VAR_OUTPUT
LampStop   :BOOL := FALSE; (* Флаг "Активен режим СТОП". *)
LampManual :BOOL := FALSE; (* Флаг "Активен РУЧНОЙ режим". *)
LampAuto   :BOOL := FALSE; (* Флаг "Активен АВТОМАТИЧЕСКИЙ режим. *)
END_VAR

VAR
State1    :INT  := 0    ; (* Локальный граф состояний. *)
FlagError :BOOL := FALSE; (* Флаг запрещенного состояния входов. *)
END_VAR

VAR CONSTANT
STATE_STOP   :INT := 0; (* Состояние "СТОП РЕЖИМ". *)
STATE_MANUAL :INT := 1; (* Состояние "РУЧНОЙ РЕЖИМ". *)
STATE_AUTO   :INT := 2; (* Состояние "АВТОМАТИЧЕСКИЙ РЕЖИМ". *)
END_VAR
(*
 Переключатель режимов работы.
          DbModeSelector
    +------------------------+
    |     FbModeSelector     |
 ->-|ButtonStop      LampStop|->-
 ->-|ButtonManual  LampManual|->-
 ->-|ButtonAuto      LampAuto|->-
   -|Error                   |
   -|Reset                   |
    +------------------------+
*)

(* Запрещенное состояние: *)
(* Если вместе с кнопкой стоп одновременно нажали еще что-то. *)
FlagError:=
((ButtonStop AND ButtonAuto) OR
( ButtonStop AND ButtonManual));

(* При перезагрузке контроллера режим СТОП. *)
IF (Reset OR FlagError) THEN
    State1     := STATE_STOP;
    LampStop   := TRUE;
    LampManual := FALSE;
    LampAuto   := FALSE;
ELSE
    (* Граф состояний. *)
    CASE State1 OF

    STATE_STOP: (* Режим СТОП. *)
    LampStop   := TRUE;
    LampManual := FALSE;
    LampAuto   := FALSE;
    (* Переход СТОП -> РУЧНОЙ. *)
    IF ButtonManual THEN
    State1     := STATE_MANUAL;
    LampStop   := FALSE;
    LampManual := TRUE;
    LampAuto   := FALSE;
    END_IF;
    (* Переход СТОП -> АВТОМАТ. *)
    IF (ButtonAuto AND NOT(Error)) THEN
    State1     := STATE_AUTO;
    LampStop   := FALSE;
    LampManual := FALSE;
    LampAuto   := TRUE;
    END_IF;

    STATE_MANUAL: (* Режим РУЧНОЙ. *)
    LampStop   := FALSE;
    LampManual := TRUE;
    LampAuto   := FALSE;
    (* Переход РУЧНОЙ -> СТОП. *)
    IF ButtonStop THEN
    State1     := 0;
    LampStop   := TRUE;
    LampManual := FALSE;
    LampAuto   := FALSE;
    END_IF;
    (* Преход РУЧНОЙ -> АВТОМАТ. *)
    IF (ButtonAuto AND NOT(Error)) THEN
    State1     := STATE_AUTO;
    LampStop   := FALSE;
    LampManual := FALSE;
    LampAuto   := TRUE;
    END_IF;

    STATE_AUTO: (* Режим АВТОМАТ. *)
    LampStop   := FALSE;
    LampManual := FALSE;
    LampAuto   := TRUE;
    (* Переход АВТОМАТ -> СТОП. *)
    IF (ButtonStop OR Error) THEN
    State1     := STATE_STOP;
    LampStop   := TRUE;
    LampManual := FALSE;
    LampAuto   := FALSE;
    END_IF;
    (* Переход АВТОМАТ -> РУЧНОЙ. *)
    IF ButtonManual THEN
    State1     := STATE_MANUAL;
    LampStop   := FALSE;
    LampManual := TRUE;
    LampAuto   := FALSE;
    END_IF;

    ELSE (*СТОП при неопределенном состоянии. *)
    State1 := STATE_STOP;
    END_CASE;

END_IF; (* IF (Reset OR FlagError) THEN *)

(*
 Граф состояний.

 Если ошибка Error активна можно работать только в ручном режиме.
 Reset должен срабатывать при перезагрузке или включении питания.

                                  |
                                 -+-Reset OR FlagError
                                  |
                                  V
                        +-------------------+
                        | State1 =          |
            +---------->| STATE_STOP        |-----------+
            |           | LampStop = 1      |           |
            |           +-------------------+           |
            |                |         ^                |
            |                |         |                |
            |   ButtonManual-+-       -+-ButtonStop     |
            |                |         |                |
            |                V         |                |
            |           +-------------------+           |
 ButtonStop |           | State1 =          |           | ButtonAuto
        OR -+-          | STATE_MANUAL      |          -+- AND
      Error |           | LampManual = 1    |           | NOT(Error)
            |           +-------------------+           |
            |                |         ^                |
            |     ButtonAuto |         |                |
            |           AND -+-       -+-ButtonManual   |
            |     NOT(Error) |         |                |
            |                V         |                |
            |           +-------------------+           |
            |           | State1 =          |           |
            +-----------| STATE_AUTO        |<----------+
                        | LampAuto = 1      |
                        +-------------------+

 Пример организации интерфейса пользователя для HMI.
 При нажатии кнопоки AUTO тег ButtonAuto = 1.
 В автоматическом режиме работы тег LampAuto = 1 дает эффект нажатия на кнопку AUTO.
 Кнопки MANUAL, STOP работают аналогично.
 Так как кнопки без фиксации то можно параллельно кнопкам на экране подключать физические кнопки.

 +--------------------------------------------------------+
 | MENU: "Errors"                                         |
 +--------------------------------------------------------+
 | 0. No Error (OK).                                      |
 |                                                        |
 |                                                        |
 |                                                        |
 |                                                        |
 |                                                        |
 |                                                        |
 +--------------------------------------------------------+
 | +--------+ +--------+ +--------+ +--------+ +--------+ |
 | | < MENU | |  AUTO  | | MANUAL | |  STOP  | | MENU > | |
 | +--------+ +--------+ +--------+ +--------+ +--------+ |
 +--------------------------------------------------------+

@COPYLEFT ALL WRONGS RESERVED :)
Author: VA
Contacts: DIY.PLC.314@gmail.com
Date start LIB_PLC: 2014
License: GNU GPL-2.0-or-later
https://www.gnu.org/licenses/old-licenses/gpl-2.0.html
https://www.youtube.com/watch?v=n1F_MfLRlX0
https://www.youtube.com/@DIY_PLC
https://github.com/DIYPLC/LIB_PLC
https://oshwlab.com/diy.plc.314/PLC_HW1_SW1
https://3dtoday.ru/3d-models/mechanical-parts/body/korpus-na-din-reiku
https://t.me/DIY_PLC
*)
END_FUNCTION_BLOCK

(* POU LIB_PLC/FbMotor, ST *)
FUNCTION_BLOCK FbMotor (* Двигатель с частотником и контактором. *)

VAR_INPUT
MotorRun       :BOOL := FALSE; (* Команда: включить двигатель. *)
VoltageOk      :BOOL := FALSE; (* Схема собрана 380VAC Ok. *)
DriveOk        :BOOL := FALSE; (* Обратная связь: нет ошибок на частотном приводе. *)
ContactorOk    :BOOL := FALSE; (* Обратная связь: контактор включился. *)
TimeMonitoring :DINT := 1000 ; (* Время гарантированного включения контактора [мс]. *)
TimeDelayOn    :DINT := 1000 ; (* Время задержки включения частотника [мс]. *)
TimeDelayOff   :DINT := 5000 ; (* Время задержки выключения контактора [мс]. *)
Ts_ms          :DINT := 100  ; (* Шаг дискретизации по времени [мс]. *)
Reset          :BOOL := FALSE; (* Сброс при перезагрузке. *)
END_VAR

VAR_OUTPUT
MotorOn        :BOOL := FALSE; (* Включить двигатель. *)
ContactorOn    :BOOL := FALSE; (* Включить контактор. *)
ErrorVoltage   :BOOL := FALSE; (* Схема разобрана нет 380VAC. *)
ErrorDrive     :BOOL := FALSE; (* Ошибка частотного привода. *)
ErrorContactor :BOOL := FALSE; (* Ошибка контактора. *)
END_VAR

VAR
State1 :INT  := 0; (* Граф сосояния частотника и контактора. *)
Timer1 :DINT := 0; (* Таймер для задержки переключения между частотником и контактором [мс]. *)
Timer2 :DINT := 0; (* Таймер для формирования ошибки контактора [мс]. *)
END_VAR

VAR CONSTANT
STATE_STOP          :INT := 0; (* Состояние "Стоп". *)
STATE_CONTACTOR_ON  :INT := 1; (* Состояние "Включение контактора". *)
STATE_DRIVE_ON      :INT := 2; (* Состояние "Включение частотного привода". *)
STATE_RUN           :INT := 3; (* Состояние "Работа". *)
STATE_DRIVE_OFF     :INT := 4; (* Состояние "Выключение частотного привода". *)
STATE_CONTACTOR_OFF :INT := 5; (* Состояние "Выключение контактора". *)
END_VAR
(*
 Двигатель с частотником и контактором.
                 DbMotor
    +-------------------------------+
    |            FbMotor            |
 ->-|MotorRun                MotorOn|->-
   -|VoltageOk           ContactorOn|-
   -|DriveOk            ErrorVoltage|-
   -|ContactorOk          ErrorDrive|-
   -|TimeMonitoring   ErrorContactor|-
   -|TimeDelayOn                    |
   -|TimeDelayOff                   |
   -|Ts_ms                          |
   -|Reset                          |
    +-------------------------------+
*)

(* Схема разобрана нет 380VAC. *)
ErrorVoltage := NOT(VoltageOk);

(* Ошибка частотного привода. *)
ErrorDrive := NOT(DriveOk);

(* Формируем ошибку контактора. *)
(* Контактор включается не сразу. *)
(* За время TimeMonitoring контактор обязан включиться, иначе ошибка. *)
(* Так же следим чтобы контактор выключился и контакты не залипли. *)
IF (ContactorOn) THEN
(* Следим чтобы контактор вовремя включился. *)
  IF (ContactorOk) THEN
  (* Контактор включился. *)
  Timer2 := 0;
  ErrorContactor := FALSE;
  ELSE
    IF (Timer2 <= TimeMonitoring) THEN
    (* Контактор еще не включился. *)
    Timer2 := Timer2 + Ts_ms;
    ErrorContactor := FALSE;
    ELSE
    (* Ошибка контактор не включился за время TimeMonitoring *)
    ErrorContactor := TRUE;
    END_IF;
  END_IF;
ELSE
(* Следим чтобы контактор вовремя выключился. *)
  IF NOT(ContactorOk) THEN
  (* Контактор выключился. *)
  Timer2 := 0;
  ErrorContactor := FALSE;
  ELSE
    IF (Timer2 <= TimeMonitoring) THEN
    (* Контактор еще не выключился. *)
    Timer2 := Timer2 + Ts_ms;
    ErrorContactor := FALSE;
    ELSE
    (* Ошибка контактор не выключился за время TimeMonitoring *)
    ErrorContactor := TRUE;
    END_IF;
  END_IF;
END_IF;

(* Сброс при перезагрузке или ошибке. *)
IF (Reset OR ErrorVoltage OR ErrorDrive) THEN
State1 := STATE_STOP;
END_IF;

(* При включении двигателя должен сначала включиться контактор затем частотный привод. *)
(* При выключении двигателя должен сначала выключиться частотный привод, а затем контактор. *)
(* Это необходимо для увеличения времени жизни контактора. *)
(* Граф состояний. *)
CASE State1 OF

(* Состояние "Стоп". *)
STATE_STOP:
MotorOn     := FALSE;
ContactorOn := FALSE;
Timer1 := 0;
(* Если получили разрешение на включение то включаем контактор. *)
IF (MotorRun) THEN
State1 := STATE_CONTACTOR_ON;
END_IF;

(* Состояние "Включение контактора". *)
STATE_CONTACTOR_ON:
MotorOn     := FALSE;
ContactorOn := TRUE;
Timer1 := Timer1 + Ts_ms;
(* Перед включением частотника делаем паузу чтоб контактор успел включиться. *)
IF (Timer1 >= TimeDelayOn) THEN
State1 := STATE_DRIVE_ON;
END_IF;

(* Состояние "Включение частотного привода". *)
STATE_DRIVE_ON:
MotorOn     := TRUE;
ContactorOn := TRUE;
Timer1 := 0;
State1 := STATE_RUN;

(* Состояние "Работа". *)
STATE_RUN:
MotorOn     := TRUE;
ContactorOn := TRUE;
Timer1 := 0;
(* Если пришла команда выключить двигатель то сначала выключаем частотник. *)
IF NOT(MotorRun) THEN
State1 := STATE_DRIVE_OFF;
END_IF;

(* Состояние "Выключение частотного привода". *)
STATE_DRIVE_OFF:
MotorOn     := FALSE;
ContactorOn := TRUE;
Timer1 := Timer1 + Ts_ms;
(* Перед выключением контактора делаем паузу чтоб выключится без нагрузки. *)
IF (Timer1 >= TimeDelayOff) THEN
State1 := STATE_CONTACTOR_OFF;
END_IF;

(* Состояние "Выключение контактора". *)
STATE_CONTACTOR_OFF:
MotorOn     := FALSE;
ContactorOn := FALSE;
Timer1 := 0;
(* Переходим в состояние стоп. *)
State1 := STATE_STOP;

(* СТОП при неопределенном состоянии. *)
ELSE
State1 := STATE_STOP;
END_CASE;

(*
 Схема подключения блока FbMotor.

                +-------------------+
                | 380 VAC           |
                +-------------------+
                          |
                          v
                +-------------------+
                | Вводной автомат   |--> VoltageOk
                +-------------------+
                          |
                          v
                +-------------------+
     MotorOn -->| Частотный привод  |--> DriveOk
                +-------------------+
                          |
                          v
                +-------------------+
 ContactorOn -->| Контактор         |--> ContactorOk
                +-------------------+
                          |
                          v
                +-------------------+
                | Двигатель         |
                +-------------------+

@COPYLEFT ALL WRONGS RESERVED :)
Author: VA
Contacts: DIY.PLC.314@gmail.com
Date start LIB_PLC: 2014
License: GNU GPL-2.0-or-later
https://www.gnu.org/licenses/old-licenses/gpl-2.0.html
https://www.youtube.com/watch?v=n1F_MfLRlX0
https://www.youtube.com/@DIY_PLC
https://github.com/DIYPLC/LIB_PLC
https://oshwlab.com/diy.plc.314/PLC_HW1_SW1
https://3dtoday.ru/3d-models/mechanical-parts/body/korpus-na-din-reiku
https://t.me/DIY_PLC
*)
END_FUNCTION_BLOCK

(* POU LIB_PLC/FbPIDstep, ST *)
FUNCTION_BLOCK FbPIDstep (* ПИД-регулятор с двумя дискретными выходами. *)

VAR_INPUT
	PV       :REAL := 0.0  ; (* Измеренное значение регулируемого параметра 0...100[%]. *)
	SP       :REAL := 0.0  ; (* Заданное значение регулируемого параметра 0...100[%]. *)
	COM_RST  :BOOL := FALSE; (* Полная перезагрузка. *)
	LMNR_HS  :BOOL := FALSE; (* Датчик обранной связи клапан открыт. *)
	LMNR_LS  :BOOL := FALSE; (* Датчик обранной связи клапан закрыт. *)
	LMNS_ON  :BOOL := FALSE; (* Включить ружной режим управления. *)
	LMNUP    :BOOL := FALSE; (* Команда открыть в ручном режиме. *)
	LMNDN    :BOOL := FALSE; (* Команда закрыть в ручном режиме. *)
	GAIN     :REAL := 2.0  ; (* Пропорциональное усиление ошибки регулирования. *)
	TI       :REAL := 20.0 ; (* Время интегрирования [с]. *)
	DEADB_W  :REAL := 0.5  ; (* Зона нечувствительности к ошибке регулирования [%]. *)
	PULSE_TM :REAL := 1.0  ; (* Минимальное время выходного импульса [с]. *)
	BREAK_TM :REAL := 1.0  ; (* Минимально время между выходными импульсами [с]. *)
	MTR_TM   :REAL := 55.0 ; (* Время открытия исполнительного механизма с 0 до 100 [с]. *)
	DISV     :REAL := 0.0  ; (* Возмущающее воздействие к ошибке регулирования [%]. *)
	CYCLE    :REAL := 0.1  ; (* Шаг дискретизации по времени [с]. *)
END_VAR

VAR_OUTPUT
	QLMNUP :BOOL :=  FALSE; (* Открыть задвижку. *)
	QLMNDN :BOOL :=  FALSE; (* Закрыть задвижку. *)
END_VAR

VAR
	ER          :REAL := 0.0  ; (* Ошибка регулирования [%]. *)
	LMNRS_ON    :BOOL := FALSE; (* *)
	LMNRSVAL    :REAL := 0.0  ; (* *)
	LMNR_SIM    :REAL := 0.0  ; (* *)
	sFbPVal     :REAL := 0.0  ; (* Меняется во время регулирования. *)
	sThrOn      :REAL := 0.0  ; (* Иногда меняется во время регулирования (похоже на адаптивный гистерезис). *)
	siImpAus    :INT  := 0    ; (* -100...0...+100 *)
	stImpDauer  :REAL := 0.0  ; (* *)
	stPausDauer :REAL := 0.0  ; (* *)
END_VAR

VAR_TEMP
	Hvar     :REAL := 0.0 ; (* Вспомогательная переменная *)
	ErKp     :REAL := 0.0 ; (* Вспомогательная переменная *)
	rTi      :REAL := 0.0 ; (* Время интегрирования в real !!! не удалять !!! *)
	AdapIn1  :REAL := 0.0 ; (* Eingang 1 der Adaption der Ansprechschwelle *)
	AdapIn2  :REAL := 0.0 ; (* Eingang 2 der Adaption der Ansprechschwelle *)
	iImpEin  :INT  := 0   ; (* Eingang des Impulsformers *)
	rThrOff  :REAL := 0.0 ; (* Abschaltschwelle *)
	dInteg   :REAL := 0.0 ; (* Eingang des Integrierers in der Rückführung *)
	dThrStIn :REAL := 0.0 ; (* Three - step element input *)
	LmnrSim  :REAL := 0.0 ; (* Simulierte Stellungsrückmeldung *)
END_VAR
(*
 ПИД-регулятор с двумя дискретными выходами.
             DbPIDstep
    +-------------------------+
    |        FbPIDstep        |
 ->-|PV                 QLMNUP|->-
   -|SP                 QLMNDN|->-
   -|COM_RST                  |
   -|LMNR_HS                  |
   -|LMNR_LS                  |
   -|LMNS_ON                  |
   -|LMNUP                    |
   -|LMNDN                    |
   -|GAIN                     |
   -|TI                       |
   -|DEADB_W                  |
   -|PULSE_TM                 |
   -|BREAK_TM                 |
   -|MTR_TM                   |
   -|DISV                     |
   -|CYCLE                    |
    +-------------------------+
*)

IF COM_RST
THEN 
    LMNR_SIM    := LMNRSVAL;
    QLMNUP      := 0       ;
    QLMNDN      := 0       ;
    PV          := 0.0     ;
    ER          := 0.0     ;
    LMNRS_ON    := 0       ;
    LMNRSVAL    := 0.0     ;
    LMNR_SIM    := 0.0     ;
    sFbPVal     := 0.0     ;
    sThrOn      := 0.0     ;
    siImpAus    := 0       ;
    stImpDauer  := 0.0     ;
    stPausDauer := 0.0     ;
ELSE
    ErKp := SP - PV;
    IF    ErKp < ( -DEADB_W) THEN  ER := ErKp + DEADB_W;
    ELSIF ErKp > DEADB_W      THEN  ER := ErKp - DEADB_W;
    ELSE  ER := 0.0; END_IF;
    ErKp := ER * GAIN;
    rTi := TI;
    IF rTi < CYCLE * 0.5 THEN rTi := CYCLE * 0.5; END_IF; 
    Hvar := rTi - ABS(0.01 * ErKp * MTR_TM);
    IF Hvar < (rTi * 0.1)THEN rTi := rTi * 0.1; ELSE rTi := Hvar; END_IF;
    IF LMNS_ON 
    THEN 
        sFbPVal := 0.0;
    ELSE  
        IF siImpAus <> 0 
        THEN  
            dInteg := DINT_TO_REAL(INT_TO_DINT(siImpAus)) * CYCLE / MTR_TM;
        ELSE 
            IF (ErKp > 0.0 AND LMNR_HS) OR (ErKp < 0.0 AND LMNR_LS) OR (TI = 0.0)
            THEN 
                dInteg := 0.0;
            ELSE    
                dInteg  := (-ErKp) * CYCLE / rTi;
            END_IF;
        END_IF;
        sFbPVal := sFbPVal + dInteg;
        IF TI = 0.0
        THEN  
            IF    sFbPVal > 100.0 THEN sFbPVal := 100.0;
            ELSIF sFbPVal < 0.0   THEN sFbPVal := 0.0;
            END_IF;
        END_IF;
    END_IF;
    dThrStIn := ErKp - sFbPVal + DISV;
    AdapIn1 := ErKp;
    AdapIn2 := sFbPVal;
    rThrOff := 55.0 / MTR_TM * CYCLE;
    IF PULSE_TM > CYCLE
    THEN
    Hvar := PULSE_TM;
    ELSE
    Hvar := CYCLE;
    END_IF;
    Hvar := 100.0 * Hvar / MTR_TM;
    IF NOT(LMNR_HS OR LMNR_LS)
    THEN
        IF NOT (QLMNUP OR QLMNDN)
        THEN
            IF TI <> 0.0
            THEN
                IF ABS(AdapIn1) < ABS(AdapIn2)
                THEN
                    sThrOn := AdapIn1;
                ELSE
                    sThrOn := AdapIn2; 
                END_IF;
            ELSE
                IF PV = 0.0
                THEN
                    sThrOn := Hvar;
                ELSE 
                    sThrOn := ABS(ErKp) * 0.5;
                END_IF;
            END_IF;
            IF sThrOn > 10.0 THEN sThrOn := 10.0; END_IF;
            IF sThrOn < Hvar THEN sThrOn := Hvar; END_IF;
        END_IF;
    ELSE
        sThrOn := Hvar;
    END_IF;
    IF (siImpAus = 100 AND dThrStIn > rThrOff) OR (dThrStIn >= sThrOn)             THEN iImpEin := 100;
    ELSIF (siImpAus = -100 AND dThrStIn < ( -rThrOff)) OR (dThrStIn <= ( -sThrOn)) THEN iImpEin := -100;
    ELSE                                                                                iImpEin := 0;
    END_IF;
    IF LMNS_ON
    THEN
        IF LMNUP XOR LMNDN
        THEN
            IF LMNUP
            THEN
                iImpEin := 100;
            ELSE
                iImpEin := -100;
            END_IF;
        ELSE
            iImpEin := 0;
        END_IF;
    END_IF;
    IF (iImpEin = 100 AND LMNR_HS) OR (iImpEin = -100 AND LMNR_LS) THEN iImpEin := 0; END_IF;
    IF (siImpAus = -100 AND iImpEin = 100) OR (siImpAus = 100 AND iImpEin = -100)THEN iImpEin := 0; END_IF;
    IF siImpAus <> iImpEin
    THEN
        IF iImpEin = 0
        THEN
            IF stImpDauer <= 0.0
            THEN 
                siImpAus := 0;
                stPausDauer := BREAK_TM;
            END_IF;
        ELSE
            siImpAus := iImpEin;
            stImpDauer := PULSE_TM;
        END_IF;
    END_IF;
    IF stImpDauer > 0.0
    THEN
    stImpDauer := stImpDauer - CYCLE;
    ELSE
    stImpDauer := 0.0;
    END_IF;
    IF stPausDauer > 0.0
    THEN
    stPausDauer := stPausDauer - CYCLE;
    ELSE
    stPausDauer := 0.0;
    END_IF;
    IF ((siImpAus = 100) AND LMNR_HS) OR ((siImpAus = -100) AND LMNR_LS)
    THEN 
      siImpAus := 0;
      stImpDauer := 0.0;
    END_IF;
    IF NOT LMNRS_ON
    THEN
        LmnrSim := LMNRSVAL;
    ELSE
        LmnrSim := DINT_TO_REAL(INT_TO_DINT(siImpAus)) * CYCLE / MTR_TM + LMNR_SIM;
        IF LmnrSim >= 100.0
        THEN
            LmnrSim := 100.0;
        ELSIF  LmnrSim <= 0.0
        THEN
            LmnrSim := 0.0;
        END_IF;
    END_IF;
    LMNR_SIM := LmnrSim;
    IF siImpAus = 0
    THEN
        QLMNUP := 0;
        QLMNDN := 0;
    ELSIF siImpAus = 100
    THEN 
        QLMNUP := 1;
        QLMNDN := 0;
    ELSE 
        QLMNUP := 0;
        QLMNDN := 1;
    END_IF;
END_IF;

(*
src CONT_S FB42
reversed by komatic
cross platforms by VA
https://web.archive.org/web/20220322202418/http://plc4good.org.ua/view_post.php?id=65
https://github.com/komatic1/SCL_regulation_control/blob/main/CONT_S.scl

Добавлен: 1exan    Дата: 2020-04-26

В этом месте есть отличия от TCONT и там похоже реализация более правильная:
Здесь:
IF iImpEin=0
THEN
IF stImpDauer<=T#0MS
THEN
siImpAus:=0;
stPausDauer:=BREAK_TM;
END_IF;
ELSE
siImpAus:=iImpEin;
stImpDauer:=PULSE_TM;
END_IF;
В TCONT:
IF iImpEin = 0 THEN
IF stImpDauer <= 0.0 THEN
siImpAus := 0 ; stPausDauer := BREAK_TM ;
END_IF ;
ELSIF stPausDauer <= 0.0 THEN
siImpAus := iImpEin ; stImpDauer := PULSE_TM ; END_IF ;

Добавлен: 1exan    Дата: 2020-04-26

Конкретно вот эта строка:
ELSIF stPausDauer <= 0.0 (или T#0s) THEN
должна быть вместо простого
ELSE

Добавлен: Roman    Дата: 2021-12-02

Правильные строки:
sThrOn:=ABS(AdapIn1);
sThrOn:=ABS(AdapIn2);

IF iImpEin=0
THEN
IF stImpDauer<=T#0MS
THEN
siImpAus:=0;
stPausDauer:=BREAK_TM;
END_IF;
ELSE IF stPausDauer<=T#0MS
THEN
siImpAus:=iImpEin;
stImpDauer:=PULSE_TM;
END_IF; END_IF;

@COPYLEFT ALL WRONGS RESERVED :)
Author: VA
Contacts: DIY.PLC.314@gmail.com
Date start LIB_PLC: 2014
License: GNU GPL-2.0-or-later
https://www.gnu.org/licenses/old-licenses/gpl-2.0.html
https://www.youtube.com/watch?v=n1F_MfLRlX0
https://www.youtube.com/@DIY_PLC
https://github.com/DIYPLC/LIB_PLC
https://oshwlab.com/diy.plc.314/PLC_HW1_SW1
https://3dtoday.ru/3d-models/mechanical-parts/body/korpus-na-din-reiku
https://t.me/DIY_PLC
*)
END_FUNCTION_BLOCK

(* POU LIB_PLC/FbRamp, ST *)
FUNCTION_BLOCK FbRamp (* Рампа разгона / торможения. *)

VAR_INPUT
	In    :REAL := 0.0  ; (* Входной сигнал. *)
	Scale :REAL := 100.0; (* Диапазон времени разгона и торможения. *)
	TAcc  :REAL := 5.0  ; (* Время разгона от 0 до Scale [с]. *)
	TDec  :REAL := 5.0  ; (* Время торможения от Scale до 0 [c]. *)
	Ts    :REAL := 0.1  ; (* Шаг дискретизации по времени [с]. *)
END_VAR

VAR_OUTPUT
	Out :REAL := 0.0; (* Выходной сигнал. *)
END_VAR

VAR_TEMP
	AccMode :BOOL := FALSE; (* Активен режим ускорения. *)
	DecMode :BOOL := FALSE; (* Активен режим замедления. *)
END_VAR
(*
 Рампа разгона / торможения.
         DbRamp
    +--------------+
    |    FbRamp    |
 ->-|In         Out|->-
   -|Scale         |
   -|TAcc          |
   -|TDec          |
   -|Ts            |
    +--------------+
*)

(* Режим байпаса интегратора рампы с безударным переходом. *)
IF (Scale <= 0.0) THEN
    Out := In;
ELSE (* Штатный режим работы. *)

    (* Состояние Out до отработки шага интегрирования. *)
    (* Оптимизировать и переместить сравнения нельзя. *)
    AccMode := (In > Out); (* Активен режим ускорения. *)
    DecMode := (In < Out); (* Активен режим замедления. *)

    (* Режим ускорения рампы. *)
    IF (AccMode) THEN
        IF (TAcc <= 0.0) THEN
        Out := In;
        ELSE
        Out := Out + ((Ts * Scale) / TAcc);
        END_IF;
    END_IF;

    (* Режим замедления рампы. *)
    IF (DecMode) THEN
        IF (TDec <= 0.0) THEN
        Out := In;
        ELSE
        Out := Out - ((Ts * Scale) / TDec);
        END_IF;
    END_IF;

    (* Установившийся режим рампы. *)
    (* Состояние Out после отработки шага интегрирования. *)
    IF ( ((AccMode) AND (Out >= In))
      OR ((DecMode) AND (Out <= In))
      OR (In = Out) ) THEN
    Out := In;
    END_IF;

END_IF;

(*
 Пример использования №1.
 Скорость открытия парового клапана от 0 до 100 процентов за 90  секунд.
 Скорость закрытия парового клапана от 100 до 0 процентов за 150 секунд.
 Параметры рампы для решения этой задачи:
 DbRamp1.Scale := 100.0; //Диапазон времени разгона и торможения.
 DbRamp1.TAcc  := 90.0 ; //Время разгона от 0 до Scale [с].
 DbRamp1.TDec  := 150.0; //Время торможения от Scale до 0 [c].

 Пример использования №2.
 Скорость разгона частотного привода от 0 до 50 Герц за 20 секунд.
 Скорость торможения частотного привода от 50 до 0 Герц за 15 секунд. 
 Параметры рампы для решения этой задачи:
 DbRamp2.Scale := 50.0; //Диапазон времени разгона и торможения.
 DbRamp2.TAcc  := 20.0; //Время разгона от 0 до Scale [с].
 DbRamp2.TDec  := 15.0; //Время торможения от Scale до 0 [c].

 Пример использования №3.
 Необходимо отключть рампу и передать сигнал напрямую с входа на выход. 
 Параметры рампы для решения этой задачи:
 DbRamp3.Scale := 0.0; //Диапазон времени разгона и торможения.

 Временная характеристика.

 ^ In
 |
 100 *************
 |   *           *
 |   *           *
 |   *           *
 0---------------------------------> t[s]

 ^ Out
 |
 |   TAcc         TDec
 |    10s          5s
 |  <----->       <-->
 100       *******     ^
 |       *        *    | Scale 100%
 |     *           *   |
 |   *              *  v
 0---------------------------------> t[s]

 Угол наклона рампы.
 tg(a) = Scale / TAcc


 Блок схема.

 Константы    Переключатель    Интегратор
 +-------+     +-----------+
 | Scale |     | In > Out  |
 | ----- |-->--|--+        |
 | TAcc  |     |   \       |
 +-------+     |    \      |
               |     \     |
 +-------+     |      \    |     +-----+
 |       |     |       \   |     |  1  |
 |   0   |-->--|--+     +--|-->--| --- |-->-- Out
 |       |     | In ~= Out |     |  s  |
 +-------+     |           |     +-----+
               |           |
 +-------+     |           |
 | Scale |     |           |
 | ----- |-->--|--+        |
 | TDec  |     | In < Out  |
 +-------+     +-----------+

@COPYLEFT ALL WRONGS RESERVED :)
Author: VA
Contacts: DIY.PLC.314@gmail.com
Date start LIB_PLC: 2014
License: GNU GPL-2.0-or-later
https://www.gnu.org/licenses/old-licenses/gpl-2.0.html
https://www.youtube.com/watch?v=n1F_MfLRlX0
https://www.youtube.com/@DIY_PLC
https://github.com/DIYPLC/LIB_PLC
https://oshwlab.com/diy.plc.314/PLC_HW1_SW1
https://3dtoday.ru/3d-models/mechanical-parts/body/korpus-na-din-reiku
https://t.me/DIY_PLC
*)
END_FUNCTION_BLOCK

(* POU LIB_PLC/FbScale, ST *)
FUNCTION_BLOCK FbScale (* Масштабирование InMin...InMax -> OutMin...OutMax. *)

VAR_INPUT
	In     :REAL:= 0.0    ; (* Вход до масштабирования. *)
	InMax  :REAL:= 27648.0; (* Максимум входного диапазона. *)
	InMin  :REAL:= 0.0    ; (* Минимум входного диапазона. *)
	OutMax :REAL:= 20.0   ; (* Максимум выходного диапазона. *)
	OutMin :REAL:= 4.0    ; (* Минимум выходного диапазона. *)
END_VAR

VAR_OUTPUT
	Out :REAL := 0.0; (* Выход после масштабирования. *)
END_VAR
(*
 Масштабирование InMin...InMax -> OutMin...OutMax.
       DbScale
    +-----------+
    |  FbScale  |
 ->-|In      Out|->-
   -|InMax      |
   -|InMin      |
   -|OutMax     |
   -|OutMin     |
    +-----------+
*)

(* Масштабирование сигнала. *)
IF (InMax = InMin) THEN (* Деление на 0 может остановить процессор. *)
(* При ошибке исходных данных. *)
Out := 0.0;
ELSE
(* Масштабирование. *)
Out := (OutMax - OutMin) * ((In - InMin)/(InMax - InMin)) + OutMin;
END_IF;

(*
 Статическая характеристика.

       ^ Out
       |
 OutMax|<---------------*
       |              * |
       |            *   |
    Out|<---------*     |
       |        * |     |
       |      *   |     |
 OutMin|<---*     |     |
       |    |     |     |
       |    |     |     |
       +---------------------> In
          InMin  In   InMax

 Выход сигнал
 Out = k * In + b

 Для расчета k, b надо решить систему двух линейных уравнений с двумя неизвестными.
 {OutMax = k * InMax + b
 {OutMin = k * InMin + b

 Усиление:
      OutMax - OutMin 
 k = -----------------
       InMax - InMin  

 Смещение:
 b = OutMax - k * InMax

 После подстановки в уравнение Out = k * In + b констант k, b,
 и сокращения числа арифметических операций до минимума получаем:
 Out := (OutMax - OutMin) * ((In - InMin)/(InMax - InMin)) + OutMin;

 Данное линейное преобразование на практике легко вывести через промежуточный диаппазон 0...1:
 InMin...InMax -> 0...(InMax-InMin) -> 0...1 -> 0...(OutMax-OutMin) -> OutMin...OutMax.
 Пример рассчета давления с датчика  4...20мА -> 0...10Бар.
 4...20 -  4 = 0...16
 0...16 / 16 = 0...1
 0...1  * 10 = 0...10
 При токе 12мА
 12  -   4 = 8
 8   /  16 = 0.5
 0.5 *  10 = 5Бар
 Давление 5Бар.

@COPYLEFT ALL WRONGS RESERVED :)
Author: VA
Contacts: DIY.PLC.314@gmail.com
Date start LIB_PLC: 2014
License: GNU GPL-2.0-or-later
https://www.gnu.org/licenses/old-licenses/gpl-2.0.html
https://www.youtube.com/watch?v=n1F_MfLRlX0
https://www.youtube.com/@DIY_PLC
https://github.com/DIYPLC/LIB_PLC
https://oshwlab.com/diy.plc.314/PLC_HW1_SW1
https://3dtoday.ru/3d-models/mechanical-parts/body/korpus-na-din-reiku
https://t.me/DIY_PLC
*)
END_FUNCTION_BLOCK

(* POU LIB_PLC/FbSimMotorGear, ST *)
FUNCTION_BLOCK FbSimMotorGear (* Виртуальный МЭО для отладки шагового регулятора. *)

VAR_INPUT
CmdOpen   :BOOL := FALSE; (* Команда на открытие +. *)
CmdClose  :BOOL := FALSE; (* Команда на закрытие -. *)
TimeOpen  :REAL := 60.0 ; (* Время необходимое для открытия задвижки [с]. *)
TimeClose :REAL := 50.0 ; (* Время необходимое для закрытия задвижки [с]. *)
Ts        :REAL := 0.1  ; (* Шаг дискретизации по времени в секундах. *)
Reset     :BOOL := FALSE; (* Сброс при перезагрузке. *)
END_VAR

VAR_OUTPUT
Position    :REAL := 0.0  ; (* Положение штока 0...100 [%]. *)
SensorOpen  :BOOL := FALSE; (* Датчик на открытие задвижки. *)
SensorClose :BOOL := FALSE; (* Датчик на закрытие задвижки. *)
END_VAR

VAR_TEMP
SpeedPos :REAL := 0.0; (* Скорость открытия. *)
SpeedNeg :REAL := 0.0; (* Скорость закрытия. *)
END_VAR
(*
 Виртуальный МЭО для отладки шагового регулятора.
           DbSimMotorGear
    +--------------------------+
    |      FbSimMotorGear      |
 ->-|CmdOpen           Position|->-
 ->-|CmdClose        SensorOpen|-
   -|TimeOpen       SensorClose|-
   -|TimeClose                 |
   -|Ts                        |
   -|Reset                     |
    +--------------------------+
*)

IF(Reset) THEN
Position := 0.0;
END_IF;

SpeedPos := 100.0 / TimeOpen ; (* [%/s] *)
SpeedNeg := 100.0 / TimeClose; (* [%/s] *)

IF(CmdOpen) THEN
Position := Position + SpeedPos * Ts; (* [%] *)
END_IF;

IF(CmdClose) THEN
Position := Position - SpeedNeg * Ts; (* [%] *)
END_IF;

IF(Position >= 100.0) THEN
Position := 100.0;
SensorOpen := TRUE;
ELSE
SensorOpen := FALSE;
END_IF;

IF(Position <= 0.0) THEN
Position := 0.0;
SensorClose := TRUE;
ELSE
SensorClose := FALSE;
END_IF;

(*
@COPYLEFT ALL WRONGS RESERVED :)
Author: VA
Contacts: DIY.PLC.314@gmail.com
Date start LIB_PLC: 2014
License: GNU GPL-2.0-or-later
https://www.gnu.org/licenses/old-licenses/gpl-2.0.html
https://www.youtube.com/watch?v=n1F_MfLRlX0
https://www.youtube.com/@DIY_PLC
https://github.com/DIYPLC/LIB_PLC
https://oshwlab.com/diy.plc.314/PLC_HW1_SW1
https://3dtoday.ru/3d-models/mechanical-parts/body/korpus-na-din-reiku
https://t.me/DIY_PLC
*)
END_FUNCTION_BLOCK

(* POU LIB_PLC/FbSoftPWM, ST *)
FUNCTION_BLOCK FbSoftPWM (* ШИМ генератор двухканальный. *)

VAR_INPUT
	DutyCucle      :REAL := 50.0;   (* Коэффициент заполнения -100...0...100 [%]. *)
	PeriodPositive :REAL := 10.0;   (* Период ШИМ для положительного коэффициента заполнения [с]. *)
	PeriodNegative :REAL := 10.0;   (* Период ШИМ для отрицательного коэффициента заполнения [с]. *)
	DBMAX          :REAL := 0.001;  (* dead band - Зона нечувствительности, верхняя граница [%]. *)
	DBMIN          :REAL := -0.001; (* dead band - Зона нечувствительности, нижняя граница [%]. *)
	Ts             :REAL := 0.1;    (* Шаг дискретизации по времени [с]. *)
END_VAR

VAR_OUTPUT
	PWMPOS :BOOL := FALSE; (* Выход ШИМ для положительных значений входа. *)
	PWMNEG :BOOL := FALSE; (* Выход ШИМ для отрицательных значений входа. *)
END_VAR

VAR
	TimerPositive :REAL := 0.0; (* Таймер для положительного коэффициента заполнения [с]. *)
	TimerNegative :REAL := 0.0; (* Таймер для отрицательного коэффициента заполнения [с]. *)
END_VAR

VAR_TEMP
	Percent           :REAL := 0.0; (* Входной сигнал после зоны нечувствительности и амплитудного ограничителя -100...0...100[%]. *)
	TimePulsePositive :REAL := 0.0; (* Время импульса для положительного коэффициента заполнения [с]. *)
	TimePulseNegative :REAL := 0.0; (* Время импульса для отрицательного коэффициента заполнения [с]. *)
END_VAR
(*
 ШИМ генератор двухканальный.
            DbSoftPWM
     +---------------------+
     |      FbSoftPWM      |
  ->-|DutyCucle      PWMPOS|->-
    -|PeriodPositive PWMNEG|->-
    -|PeriodNegative       |
    -|DBMAX                |
    -|DBMIN                |
    -|Ts                   |
     +---------------------+
*)

(* Зона нечувствительности для входного сигнала. *)
IF ((DBMIN<DutyCucle)AND(DutyCucle<DBMAX)) THEN
Percent:=0.0;
ELSE
Percent:=DutyCucle;
END_IF;

(* Амплитудный ограничитель входного сигнала от -100% до 100%. *)
IF (Percent>=100.0) THEN
Percent:=100.0;
END_IF;
IF (Percent<=-100.0) THEN
Percent:=-100.0;
END_IF;

(* Формирование импульсов на открытие. *)
IF (Percent>0.0) THEN
PWMNEG:=FALSE;
TimerNegative:=0.0;
TimePulsePositive:=PeriodPositive*Percent*0.01;
    IF (TimerPositive<=TimePulsePositive) THEN
    PWMPOS:=TRUE;
    ELSE
    PWMPOS:=FALSE;
    END_IF;
TimerPositive:=TimerPositive+Ts;
    IF (TimerPositive>=PeriodPositive) THEN
    TimerPositive:=0.0;
    END_IF;
END_IF;

(* Формирование импульсов на закрытие. *)
IF (Percent<0.0) THEN
PWMPOS:=FALSE;
TimerPositive:=0.0;
TimePulseNegative:=PeriodNegative*Percent*(-0.01);
    IF (TimerNegative<=TimePulseNegative) THEN
    PWMNEG:=TRUE;
    ELSE
    PWMNEG:=FALSE;
    END_IF;
TimerNegative:=TimerNegative+Ts;
    IF (TimerNegative>=PeriodNegative) THEN
    TimerNegative:=0.0;
    END_IF;
END_IF;

(* Нет импульсов. *)
IF (Percent=0.0) THEN
PWMPOS:=FALSE;
PWMNEG:=FALSE;
TimerPositive:=0.0;
TimerNegative:=0.0;
END_IF;

(*
@COPYLEFT ALL WRONGS RESERVED :)
Author: VA
Contacts: DIY.PLC.314@gmail.com
Date start LIB_PLC: 2014
License: GNU GPL-2.0-or-later
https://www.gnu.org/licenses/old-licenses/gpl-2.0.html
https://www.youtube.com/watch?v=n1F_MfLRlX0
https://www.youtube.com/@DIY_PLC
https://github.com/DIYPLC/LIB_PLC
https://oshwlab.com/diy.plc.314/PLC_HW1_SW1
https://3dtoday.ru/3d-models/mechanical-parts/body/korpus-na-din-reiku
https://t.me/DIY_PLC
*)
END_FUNCTION_BLOCK

(* POU LIB_PLC/FbStpForPD, ST *)
FUNCTION_BLOCK FbStpForPD (* Аналоговый ПД-регулятор превращаем в дискретный ПИ. *)

VAR_INPUT
InFromPD    :REAL := 0.0  ; (* Задание скорости с обычного ПД- регулятора -100...+100 [%/c]. *)
TimeOpen    :REAL := 60.0 ; (* Время открытия задвижки [c]. *)
TimeClose   :REAL := 50.0 ; (* Время закрытия задвижки [c]. *)
TimeMin     :REAL := 0.5  ; (* Минимальное время импульса [c]. *)
Smax        :REAL := 10.0 ; (* Ограничение внутреннего интегратора положения максимум [%]. *)
Smin        :REAL := -10.0; (* Ограничение внутреннего интегратора положения минимум [%]. *)
SensorOpen  :BOOL := FALSE; (* Датчик на открытие задвижки 100 [%]. *)
SensorClose :BOOL := FALSE; (* Датчик на закрытие задвижки 0 [%]. *)
Ts          :REAL := 0.1  ; (* Шаг дискретизации по времени в секундах. *)
Reset       :BOOL := FALSE; (* Сброс при перезагрузке. *)
END_VAR

VAR_OUTPUT
CmdOpen  :BOOL := FALSE; (* Команда на открытие +. *)
CmdClose :BOOL := FALSE; (* Команда на закрытие -. *)
END_VAR

VAR
Pos :REAL := 0.0; (* Положение клапана интеграл скорости по времени есть путь [%]. *)
END_VAR

VAR_TEMP
Vin        :REAL := 0.0; (* Скорость на входе [%/с]. *)
Vopen      :REAL := 0.0; (* Скорость открытия [%/с]. *)
Vclose     :REAL := 0.0; (* Скорость закрытия [%/с]. *)
SopenMin   :REAL := 0.0; (* Минимальная дистанция доступная для перемещения на открытие[%]. *)
ScloseMin  :REAL := 0.0; (* Минимальная дистанция доступная для перемещения на закрытие[%]. *)
END_VAR
(*
 Аналоговый ПД-регулятор превращаем в дискретный ПИ.
           DbStpForPD
    +----------------------+
    |      FbStpForPD      |
 ->-|InFromPD       CmdOpen|->-
   -|TimeOpen      CmdClose|->-
   -|TimeClose             |
   -|TimeMin               |
   -|Smax                  |
   -|Smin                  |
   -|SensorOpen            |
   -|SensorClose           |
   -|Ts                    |
   -|Reset                 |
    +----------------------+
*)

(* Вычисления основаны на том, что интегрирующий исполнительный механизм работает в пределах 0...100 [%]. *)
Vin := InFromPD;               (* [%/с]. *)
Vopen  := 100.0 / TimeOpen;    (* [%/с]. *)
Vclose := 100.0 / TimeClose;   (* [%/с]. *)
SopenMin  := Vopen  * TimeMin; (* [%]. *)
ScloseMin := Vclose * TimeMin; (* [%]. *)
Pos := Pos + Vin * Ts;         (* [%]. *)

IF(Reset) THEN
Pos := 0.0;
END_IF;

(* Импульс открытия (положительный). *)
IF(Pos >= SopenMin) THEN (* RS-Триггер на открытие. *)
CmdOpen := TRUE;
END_IF;

IF((Pos <= 0.0) OR SensorOpen) THEN (* RS-Триггер на открытие. *)
CmdOpen := FALSE;
END_IF;

IF(CmdOpen) THEN (* Вход положительный итератор отрицательный. *)
Pos := Pos - Vopen * Ts; (* [%]. *)
END_IF;

(* Импульс закрытия (отрицательный). *)
IF(Pos <= (ScloseMin * (-1.0))) THEN (* RS-Триггер на закрытие. *)
CmdClose := TRUE;
END_IF;

IF((Pos >= 0.0) OR SensorClose) THEN (* RS-Триггер на закрытие. *)
CmdClose := FALSE;
END_IF;

IF(CmdClose) THEN (* Вход отрицательный интегратор положительный. *)
Pos := Pos + Vclose * Ts; (* [%]. *)
END_IF;

(* Амплитудный ограничитель интегратора. *)
IF(Pos >= Smax) THEN
Pos := Smax;
END_IF;

IF(Pos <= Smin) THEN
Pos := Smin;
END_IF;

(*
 Описание.
 Данный блок это приставка к обычному аналоговому ПИД- регулятору которая превращает его в регулятор с двумя дискретными выходами.
 Применять данный блок можно на котлах с интегральными исполнительными механизмами.
 Например, если у вас есть мотор редуктор, который управляется двумя пускателями и выходной вал имеет датчик положения и концевики положений 0% и 100%,
 то данный блок в паре с ПИД- регулятором позволит управлять положением этого механизма.
 Вместо датчика положения можно завести датчик температуры или давления и получить соответственно систему стабилизации температуры или давления.

 Основная идея данного блока состоит в том, что интегральный исполнительный механизм вместе с регулятором должен иметь передаточную функцию ПИ-регулятора.
 Из чего следует что интегральный исполнительный механизм должен управляться ПД- регулятором и тогда они вместе дадут передаточную функцию ПИ-регулятора.
 Но выход с ПД- регулятора аналоговый а исполнительный механизм дискретный.
 Так как аналоговый выход с ПД- регулятора это по сути задание скорости на интегральный исполнительный механизм, а
 дискретные сигналы это тоже суть задание положительной и отрицательной постоянной скорости,
 то остается вычислить площадь аналоговой кривой который дает ПД- регулятор, и выдать эту площадь в виде эквивалентных по площади дискретных импульсах управления.
 Другими словами можно сказать, что данный блок считает площадь сигнала произвольной формы на входе
 и выдает эквивалентную площадь дискретных сигналов на выходе с учетом его полярности.
 Так же необходимо учесть, что есть минимальное значение импульса, который может отработать исполнительный механизм.
 Еще учесть, что в общем случае, что время открытия и закрытия исполнительного механизма может быть разное.

 Изначальной данный блок планировался как самостоятельный ПИ- регулятор с двумя дискретными выходами для интегральных исполнительных механизмов.
 Но во время реализации стало понятно что более оптимально сделать приставке к обычному ПИД- регулятору который должен работать как ПД- регулятор.
 Между ПИД- регулятором и данным блоком на время отладки можно поставить дополнительный амплитудный ограничитель и зону не чувствительности.

 Данный блок проектировался ручкой в тетрадке в терминах языка CFC.
 При трансляции на структурированный текст сумматор и триггеры были реализованны не явно.

 Блок схема.

        Сумматор
          +---+    Интегратор
          |   |   +----------+
  Vopen->-|-  |   |          |
          |   |   |  Z * Ts  |
    Vin->-|+  |->-| -------- |->-S
          |   |   |  Z - 1   |
 Vclose->-|+  |   |          |
          |   |   +----------+
          +---+

 Амплитудный ограничитель
           Smax
       +-----------+
       |           |
       |       +-- |
       |      /    |
 Pos->-|     /     |->-Pos
       |    /      |
       | --+       |
       |           |
       +-----------+
           Smin

                                Триггер на открытие
                                  +-------------+
                                  | FbTriggerRS |
       +--------------+           |             |
 Pos->-| Pos >= Smin  |--------->-|Set       Out|->-CmdOpen
       +--------------+           |             |
                                  |             |
       +--------------+   +---+   |             |
 Pos->-|   Pos <= 0   |->-| 1 |->-|Rst          |
       +--------------+   |   |   |             |
                          |   |   +-------------+
             SensorOpen->-|   |
                          |   |
                          +---+

           +--------------+   +---+
 CmdOpen->-| BOOL_TO_REAL |->-| * |->-Vopen
           +--------------+   |   |
                              |   |
           100.0 / TimeOpen->-|   |
                              |   |
                              +---+

                                Триггер на закрытие
                                  +-------------+
                                  | FbTriggerRS |
       +--------------+           |             |
 Pos->-| Pos <= -Smin |--------->-|Set       Out|->-CmdClose
       +--------------+           |             |
                                  |             |
       +--------------+   +---+   |             |
 Pos->-|   Pos >= 0   |->-| 1 |->-|Rst          |
       +--------------+   |   |   |             |
                          |   |   +-------------+
            SensorClose->-|   |
                          |   |
                          +---+

            +--------------+   +---+
 CmdClose->-| BOOL_TO_REAL |->-| * |->-Vclose
            +--------------+   |   |
                               |   |
           100.0 / TimeClose->-|   |
                               |   |
                               +---+

               <-Pos->
                  |
                  V
 <----------|-----------|-----------|----------->
         -Smin          0         +Smin
        CmdClose                 CmdOpen

@COPYLEFT ALL WRONGS RESERVED :)
Author: VA
Contacts: DIY.PLC.314@gmail.com
Date start LIB_PLC: 2014
License: GNU GPL-2.0-or-later
https://www.gnu.org/licenses/old-licenses/gpl-2.0.html
https://www.youtube.com/watch?v=n1F_MfLRlX0
https://www.youtube.com/@DIY_PLC
https://github.com/DIYPLC/LIB_PLC
https://oshwlab.com/diy.plc.314/PLC_HW1_SW1
https://3dtoday.ru/3d-models/mechanical-parts/body/korpus-na-din-reiku
https://t.me/DIY_PLC
*)
END_FUNCTION_BLOCK

(* POU LIB_PLC/FbSum1bit, ST *)
FUNCTION_BLOCK FbSum1bit (* Сумматор 1бит. *)

VAR_INPUT
	A   :BOOL := FALSE; (* Первое слагаемое. *)
	B   :BOOL := FALSE; (* Второе слагаемое. *)
	Cin :BOOL := FALSE; (* Входной флаг переноса при сложении. *)
END_VAR

VAR_OUTPUT
	Sum  :BOOL := FALSE; (* Сумма. *)
	Cout :BOOL := FALSE; (* Выходной флаг переноса при сложении. *)
END_VAR
(* Сумма. *)
Sum := (NOT(A) AND NOT(B) AND Cin) OR (NOT(A) AND B AND NOT(Cin)) OR (A AND NOT(B) AND NOT(Cin)) OR (A AND B AND Cin);
(* Перенос. *)
Cout := (NOT(A) AND B AND Cin) OR (A AND NOT(B) AND Cin) OR (A AND B AND NOT(Cin)) OR (A AND B AND Cin);

(*
 Таблица истинности сумматора.
 +---+---+-----+-----+------+
 | A | B | Cin | Sum | Cout |
 +---+---+-----+-----+------+
 | 0 | 0 | 0   | 0   | 0    |
 +---+---+-----+-----+------+
 | 0 | 0 | 1   | 1   | 0    |
 +---+---+-----+-----+------+
 | 0 | 1 | 0   | 1   | 0    |
 +---+---+-----+-----+------+
 | 0 | 1 | 1   | 0   | 1    |
 +---+---+-----+-----+------+
 | 1 | 0 | 0   | 1   | 0    |
 +---+---+-----+-----+------+
 | 1 | 0 | 1   | 0   | 1    |
 +---+---+-----+-----+------+
 | 1 | 1 | 0   | 0   | 1    |
 +---+---+-----+-----+------+
 | 1 | 1 | 1   | 1   | 1    |
 +---+---+-----+-----+------+
 Получившийся сумматор состоит из 31ой элементарной операций типа И,ИЛИ,НЕ.
 Данная реализация самая наглядная но не факт, что оптимальная.
 Сумма формируется 4мя дешифраторами соединенными по схеме ИЛИ.
 Флаг переноса формируется 4мя дешифраторами соединенными по схеме ИЛИ.
 Сумматор подходит для целых 8битных чисел без знаком 0...255. (тестировано.)
 Сумматор подходит для целых 7битных чисел со знаком -127...127. (надо протестировать заем...)

********************************************************

 AND
 |    X1       X2       Y1   |
 +---| |------| |------( )---+
 |                           |

 OR
 |    X1           Y1   |
 +---| |---+------( )---+
 |         |            |
 |    X2   |            |
 +---| |---+            |
 |                      |

 NOT
 |    X1       Y1   |
 +---|/|------( )---+
 |                  |

********************************************************

        +-----+   +-----+   +----+
   A ->-| NOT |->-| AND |->-| OR |->- Sum
        +-----+   |     |   |    |
        +-----+   |     |   |    |
   B ->-| NOT |->-|     |   |    |
        +-----+   |     |   |    |
                  |     |   |    |
 Cin ->-----------|     |   |    |
                  +-----+   |    |
        +-----+   +-----+   |    |
   A ->-| NOT |->-| AND |->-|    |
        +-----+   |     |   |    |
                  |     |   |    |
   B ->-----------|     |   |    |
                  |     |   |    |
        +-----+   |     |   |    |
 Cin ->-| NOT |->-|     |   |    |
        +-----+   +-----+   |    |
                  +-----+   |    |
   A ->-----------| AND |->-|    |
                  |     |   |    |
        +-----+   |     |   |    |
   B ->-| NOT |->-|     |   |    |
        +-----+   |     |   |    |
        +-----+   |     |   |    |
 Cin ->-| NOT |->-|     |   |    |
        +-----+   +-----+   |    |
                  +-----+   |    |
   A ->-----------| AND |   |    |
                  |     |   |    |
                  |     |   |    |
   B ->-----------|     |   |    |
                  |     |   |    |
                  |     |   |    |
 Cin ->-----------|     |   |    |
                  +-----+   +----+

    +--------+
 ->-|Cin  Sum|->-
 ->-|A       |
 ->-|B       |
    +--------+

        +-----+   +-----+   +----+
   A ->-| NOT |->-| AND |->-| OR |->- Cout
        +-----+   |     |   |    |
                  |     |   |    |
   B ->-----------|     |   |    |
                  |     |   |    |
                  |     |   |    |
 Cin ->-----------|     |   |    |
                  +-----+   |    |
                  +-----+   |    |
   A ->-----------| AND |->-|    |
                  |     |   |    |
        +-----+   |     |   |    |
   B ->-| NOT |->-|     |   |    |
        +-----+   |     |   |    |
                  |     |   |    |
 Cin ->-----------|     |   |    |
                  +-----+   |    |
                  +-----+   |    |
   A ->-----------| AND |->-|    |
                  |     |   |    |
                  |     |   |    |
   B ->-----------|     |   |    |
                  |     |   |    |
        +-----+   |     |   |    |
 Cin ->-| NOT |->-|     |   |    |
        +-----+   +-----+   |    |
                  +-----+   |    |
   A ->-----------| AND |->-|    |
                  |     |   |    |
                  |     |   |    |
   B ->-----------|     |   |    |
                  |     |   |    |
                  |     |   |    |
 Cin ->-----------|     |   |    |
                  +-----+   +----+

    +--------+
 ->-|Cin Cout|->-
 ->-|A       |
 ->-|B       |
    +--------+

********************************************************

       +--------+
  0 ->-|Cin  Sum|->- Sum0
 A0 ->-|A   Cout|->-+
 B0 ->-|B       |   |
       +--------+   |
                    |
   +----------------+
   |
   |   +--------+
   +->-|Cin  Sum|->- Sum1
 A1 ->-|A   Cout|->-+
 B1 ->-|B       |   |
       +--------+   |
                    |
   +----------------+
   |
   |   +--------+
   +->-|Cin  Sum|->- Sum2
 A2 ->-|A   Cout|->-+
 B2 ->-|B       |   |
       +--------+   |
                    |
   +----------------+
   |
   |   +--------+
   +->-|Cin  Sum|->- Sum3
 A3 ->-|A   Cout|->-+
 B3 ->-|B       |   |
       +--------+   |
                    |
   +----------------+
   |
   |   +--------+
   +->-|Cin  Sum|->- Sum4
 A4 ->-|A   Cout|->-+
 B4 ->-|B       |   |
       +--------+   |
                    |
   +----------------+
   |
   |   +--------+
   +->-|Cin  Sum|->- Sum5
 A5 ->-|A   Cout|->-+
 B5 ->-|B       |   |
       +--------+   |
                    |
   +----------------+
   |
   |   +--------+
   +->-|Cin  Sum|->- Sum6
 A6 ->-|A   Cout|->-+
 B6 ->-|B       |   |
       +--------+   |
                    |
   +----------------+
   |
   |   +--------+
   +->-|Cin  Sum|->- Sum7
 A7 ->-|A   Cout|->- Cout
 B7 ->-|B       |
       +--------+

********************************************************

 AVR ASM
 LDI R16,2
 LDI R17,3
 ADD R16, R17

********************************************************

 GCC
 uint8_t add(uint8_t A, uint8_t B) {
 return (A + B); }

********************************************************

@COPYLEFT ALL WRONGS RESERVED :)
Author: VA
Contacts: DIY.PLC.314@gmail.com
Date start LIB_PLC: 2014
License: GNU GPL-2.0-or-later
https://www.gnu.org/licenses/old-licenses/gpl-2.0.html
https://www.youtube.com/watch?v=n1F_MfLRlX0
https://www.youtube.com/@DIY_PLC
https://github.com/DIYPLC/LIB_PLC
https://oshwlab.com/diy.plc.314/PLC_HW1_SW1
https://3dtoday.ru/3d-models/mechanical-parts/body/korpus-na-din-reiku
https://t.me/DIY_PLC
*)
END_FUNCTION_BLOCK

(* POU LIB_PLC/FbTOF, ST *)
FUNCTION_BLOCK FbTOF (* Таймер с задержкой на выключение. *)

VAR_INPUT
	In           :BOOL := FALSE; (* Вход таймера. *)
	TimeDelayOff :UDINT := 5000 ; (* Время задержки выключения [мс]. *)
	Ts_ms        :UDINT := 100  ; (* Шаг дискретизации по времени [мс]. *)
END_VAR

VAR_OUTPUT
	Out :BOOL := FALSE; (* Выход таймера. *)
END_VAR

VAR
	Timer1 :UDINT := 0; (* Текущее время таймер1 [мс]. *)
END_VAR
(*
 Таймер с задержкой на выключение.
          DbTOF
    +----------------+
    |     FbTOF      |
 ->-|In           Out|->-
   -|TimeDelayOff    |
   -|Ts_ms           |
    +----------------+
*)

IF (TimeDelayOff > 0) THEN (* Таймер включен. *)
  IF (In) THEN (* На входе 1 то на выходе тоже 1. *)
  Out := TRUE;
  Timer1 := 0;   
  ELSE (* Если на входе 0. *)
    IF (Out) THEN (* На выходе 1. *)
      IF (Timer1 >= TimeDelayOff) THEN (* Задержка включения закончилась. *)
      Out := FALSE;
      Timer1 := 0;
      ELSE (* Задержка включения активна. *)
      Out := TRUE;
      Timer1 := Timer1 + Ts_ms;
      END_IF;
    ELSE (* На выходе 0. *)
    Out := FALSE;
    Timer1 := 0;
    END_IF;
  END_IF;
ELSE (* Таймер выключен. *)
Out := In;
Timer1 := 0;
END_IF;

(*
 Применение.

 Блок может применятся как фильтр дребезга контактов и как расширитель импульсов.

 Временная характеристика.

  In
  ^
  |     TimeDelayOff          TimeDelayOff
  |       |<--->|               |<--->|
 1|   *****     |     ***** *** *     |
  |   *   *     |     *   * * * *     |
 0*****---*************---***-*************----> t[s]

  Out
  ^
  |     TimeDelayOff          TimeDelayOff
  |       |<--->|               |<--->|
 1|   ***********     *****************
  |   *         *     *               *
 0*****---------*******---------------*****----> t[s]

@COPYLEFT ALL WRONGS RESERVED :)
Author: VA
Contacts: DIY.PLC.314@gmail.com
Date start LIB_PLC: 2014
License: GNU GPL-2.0-or-later
https://www.gnu.org/licenses/old-licenses/gpl-2.0.html
https://www.youtube.com/watch?v=n1F_MfLRlX0
https://www.youtube.com/@DIY_PLC
https://github.com/DIYPLC/LIB_PLC
https://oshwlab.com/diy.plc.314/PLC_HW1_SW1
https://3dtoday.ru/3d-models/mechanical-parts/body/korpus-na-din-reiku
https://t.me/DIY_PLC
*)
END_FUNCTION_BLOCK

(* POU LIB_PLC/FbTON, ST *)
FUNCTION_BLOCK FbTON (* Таймер с задержкой на включение. *)

VAR_INPUT
	In          :BOOL := FALSE; (* Вход таймера. *)
	TimeDelayOn :UDINT := 5000 ; (* Время задержки включения [мс]. *)
	Ts_ms       :UDINT := 100  ; (* Шаг дискретизации по времени [мс]. *)
END_VAR

VAR_OUTPUT
	Out :BOOL := FALSE; (* Выход таймера. *)
END_VAR

VAR
	Timer1 :UDINT := 0; (* Текущее время таймер1 [мс]. *)
END_VAR
(*
 Таймер с задержкой на включение.
          DbTON
    +----------------+
    |     FbTON      |
 ->-|In           Out|->-
   -|TimeDelayOn     |
   -|Ts_ms           |
    +----------------+
*)

IF (TimeDelayOn > 0) THEN (* Таймер включен. *)
  IF (In) THEN (* На входе 1. *)
    IF (Out) THEN (* На выходе 1. *)
    Out := TRUE;
    Timer1 := 0;
    ELSE (* На выходе 0. *)
      IF (Timer1 >= TimeDelayOn) THEN (* Задержка включения закончилась. *)
      Out := TRUE;
      Timer1 := 0;
      ELSE (* Задержка включения активна. *)
      Out := FALSE;
      Timer1 := Timer1 + Ts_ms;
      END_IF;
    END_IF;
  ELSE (* Если на входе 0 то на выходе тоже 0. *)
  Out := FALSE;
  Timer1 := 0;
  END_IF;
ELSE (* Таймер выключен. *)
Out := In;
Timer1 := 0;
END_IF;

(*
 Применение.

 При поступлении входного сигнала выходной сигнал появляется не сразу, а с задержкой TimeDelayOn.
 Блок может применятся как фильтр дребезга контактов дискретных входов.
 Совместно с инвертором может применяться для генерации импульсов.

 Временная характеристика.

  In
  ^
  | TimeDelayOn           TimeDelayOn
  |   |<--->|               |<--->|
 1|   ***********     * *   ***********
  |   *         *     * *   *         *
 0*****---------*************---------*****----> t[s]

  Out
  ^
  | TimeDelayOn           TimeDelayOn
  |   |<--->|               |<--->|
 1|   |     *****           |     *****
  |   |     *   *           |     *   *
 0***********---*******************---*****----> t[s]

@COPYLEFT ALL WRONGS RESERVED :)
Author: VA
Contacts: DIY.PLC.314@gmail.com
Date start LIB_PLC: 2014
License: GNU GPL-2.0-or-later
https://www.gnu.org/licenses/old-licenses/gpl-2.0.html
https://www.youtube.com/watch?v=n1F_MfLRlX0
https://www.youtube.com/@DIY_PLC
https://github.com/DIYPLC/LIB_PLC
https://oshwlab.com/diy.plc.314/PLC_HW1_SW1
https://3dtoday.ru/3d-models/mechanical-parts/body/korpus-na-din-reiku
https://t.me/DIY_PLC
*)
END_FUNCTION_BLOCK

(* POU LIB_PLC/FbTriggerRS, ST *)
FUNCTION_BLOCK FbTriggerRS (* RS- Триггер с приоритетом на сброс.' *)

VAR_INPUT
	Set :BOOL := FALSE; (* Set — установить единицу. *)
	Rst :BOOL := FALSE; (* Reset — сбросить на ноль. *)
END_VAR

VAR_OUTPUT
	Out :BOOL := FALSE; (* Выход триггера. *)
END_VAR
(*
 RS- Триггер с приоритетом на сброс.
       DbTriggerRS
     +-------------+
     | FbTriggerRS |
  ->-|Set       Out|->-
  ->-|Rst          |
     +-------------+
*)

(* RS- Триггер. *)
Out := (Out OR Set) AND (NOT(Rst));

(*
  Релейная интерпритация. 
 |                       |
 |  Rst     Set     Out  |
 +--|/|--+--| |--+--( )--+
 |       |       |       |
 |       |  Out  |       |
 |       +--| |--+       |
 |                       |

@COPYLEFT ALL WRONGS RESERVED :)
Author: VA
Contacts: DIY.PLC.314@gmail.com
Date start LIB_PLC: 2014
License: GNU GPL-2.0-or-later
https://www.gnu.org/licenses/old-licenses/gpl-2.0.html
https://www.youtube.com/watch?v=n1F_MfLRlX0
https://www.youtube.com/@DIY_PLC
https://github.com/DIYPLC/LIB_PLC
https://oshwlab.com/diy.plc.314/PLC_HW1_SW1
https://3dtoday.ru/3d-models/mechanical-parts/body/korpus-na-din-reiku
https://t.me/DIY_PLC
*)
END_FUNCTION_BLOCK

(* POU LIB_PLC/FbWordToBits, ST *)
FUNCTION_BLOCK FbWordToBits (* Преобразование слова в 16 бит. *)

VAR_INPUT
	In :WORD := 0; (* Входной сигнал. *)
END_VAR

VAR_OUTPUT
	Out0  :BOOL := FALSE; (* Выходной сигнал бит0. *)
	Out1  :BOOL := FALSE; (* Выходной сигнал бит1. *)
	Out2  :BOOL := FALSE; (* Выходной сигнал бит2. *)
	Out3  :BOOL := FALSE; (* Выходной сигнал бит3. *)
	Out4  :BOOL := FALSE; (* Выходной сигнал бит4. *)
	Out5  :BOOL := FALSE; (* Выходной сигнал бит5. *)
	Out6  :BOOL := FALSE; (* Выходной сигнал бит6. *)
	Out7  :BOOL := FALSE; (* Выходной сигнал бит7. *)
	Out8  :BOOL := FALSE; (* Выходной сигнал бит8. *)
	Out9  :BOOL := FALSE; (* Выходной сигнал бит9. *)
	Out10 :BOOL := FALSE; (* Выходной сигнал бит10. *)
	Out11 :BOOL := FALSE; (* Выходной сигнал бит11. *)
	Out12 :BOOL := FALSE; (* Выходной сигнал бит12. *)
	Out13 :BOOL := FALSE; (* Выходной сигнал бит13. *)
	Out14 :BOOL := FALSE; (* Выходной сигнал бит14. *)
	Out15 :BOOL := FALSE; (* Выходной сигнал бит15. *)
END_VAR
(*
 Преобразование слова в 16 бит.
      DbWordToBits
    +--------------+
    | FbWordToBits |
 ->-|In        Out0|->-
    |          Out1|->-
    |          Out2|->-
    |          Out3|->-
    |          Out4|->-
    |          Out5|->-
    |          Out6|->-
    |          Out7|->-
    |          Out8|->-
    |          Out9|->-
    |         Out10|->-
    |         Out11|->-
    |         Out12|->-
    |         Out13|->-
    |         Out14|->-
    |         Out15|->-
    +--------------+
*)

(* Логическое условие без оператора if. *)
Out0:= ((In AND 2#0000000000000001) <> 0);
Out1:= ((In AND 2#0000000000000010) <> 0);
Out2:= ((In AND 2#0000000000000100) <> 0);
Out3:= ((In AND 2#0000000000001000) <> 0);
Out4:= ((In AND 2#0000000000010000) <> 0);
Out5:= ((In AND 2#0000000000100000) <> 0);
Out6:= ((In AND 2#0000000001000000) <> 0);
Out7:= ((In AND 2#0000000010000000) <> 0);
Out8:= ((In AND 2#0000000100000000) <> 0);
Out9:= ((In AND 2#0000001000000000) <> 0);
Out10:=((In AND 2#0000010000000000) <> 0);
Out11:=((In AND 2#0000100000000000) <> 0);
Out12:=((In AND 2#0001000000000000) <> 0);
Out13:=((In AND 2#0010000000000000) <> 0);
Out14:=((In AND 2#0100000000000000) <> 0);
Out15:=((In AND 2#1000000000000000) <> 0);

(*
@COPYLEFT ALL WRONGS RESERVED :)
Author: VA
Contacts: DIY.PLC.314@gmail.com
Date start LIB_PLC: 2014
License: GNU GPL-2.0-or-later
https://www.gnu.org/licenses/old-licenses/gpl-2.0.html
https://www.youtube.com/watch?v=n1F_MfLRlX0
https://www.youtube.com/@DIY_PLC
https://github.com/DIYPLC/LIB_PLC
https://oshwlab.com/diy.plc.314/PLC_HW1_SW1
https://3dtoday.ru/3d-models/mechanical-parts/body/korpus-na-din-reiku
https://t.me/DIY_PLC
*)
END_FUNCTION_BLOCK

(* POU LIB_PLC/FbValve, ST *)
FUNCTION_BLOCK FbValve (* Пневмоцилиндр с концевиками. *)

VAR_INPUT
	CommandOpen     :BOOL := FALSE; (* Команда открыть клапан. *)
	FeedbackOpen    :BOOL := FALSE; (* Датчик обратной связи "Клапан открылся". *)
	FeedbackClose   :BOOL := FALSE; (* Датчик обратной связи "Клапан закрылся". *)
	OnFeedbackOpen  :BOOL := FALSE; (* Включить датчик обратной связи "Клапан открылся". *)
	OnFeedbackClose :BOOL := FALSE; (* Включить датчик обратной связи "Клапан закрылся". *)
	Reset           :BOOL := FALSE; (* Сброс драйвера в исходное состояние. *)
	TimeOpen        :DINT := 5000 ; (* Время открытия клапана [мс]. *)
	TimeClose       :DINT := 5000 ; (* Время закрытия клапана [мс]. *)
	Ts_ms           :DINT := 100  ; (* Шаг дискретизации по времени [мс]. *)
END_VAR

VAR_OUTPUT
	CoilOpen   :BOOL := FALSE; (* Сигнал на электромагнит "Открыть клапан". *)
	StateOpen  :BOOL := FALSE; (* Сосотение "Клапан открыт". *)
	StateClose :BOOL := FALSE; (* Сосотение "Клапан закрыт". *)
	Error      :BOOL := FALSE; (* Ошибка "Неисправность клапана". *)
END_VAR

VAR
	Timer1 :DINT := 0; (* Таймер [мс]. *)
	State1 :INT  := 0; (* Граф состояния. *)
END_VAR

VAR CONSTANT
	STATE_RESET         :INT := 0; (* Сброс алгоритма. *)
	STATE_VALVE_CLOSING :INT := 1; (* Закрытие клапана. *)
	STATE_VALVE_CLOSE   :INT := 2; (* Клапан закрыт. *)
	STATE_VALVE_OPENING :INT := 3; (* Открытие клапана. *)
	STATE_VALVE_OPEN    :INT := 4; (* Клапан открыт. *)
	STATE_ERROR_CLOSE   :INT := 5; (* Клапан не закрылся. *)
	STATE_ERROR_OPEN    :INT := 6; (* Клапан не открылся. *)
END_VAR
(*
 Пневмоцилиндр с концевиками.
                DbValve
    +-----------------------------+
    |           FbValve           |
 ->-|CommandOpen          CoilOpen|->-
   -|FeedbackOpen        StateOpen|-
   -|FeedbackClose      StateClose|-
   -|OnFeedbackOpen          Error|-
   -|OnFeedbackClose              |
   -|Reset                        |
   -|TimeOpen                     |
   -|TimeClose                    |
   -|Ts_ms                        |
    +-----------------------------+
*)

CoilOpen := CommandOpen; (* Это основная часть блока все остальное нужно для удобства использования. *)

(* Сброс алгоритма. *)
IF (Reset) THEN
State1 := STATE_RESET;
END_IF;

(* Граф состояний. *)
CASE State1 OF

STATE_RESET: (* Сброс алгоритма. *)
Timer1     := 0;
StateOpen  := FALSE;
StateClose := FALSE;
Error      := FALSE;
(* Смотрим куда надо перейти на закрытие или открытие. *)
IF (CommandOpen) THEN
State1 := STATE_VALVE_OPENING;
ELSE
State1 := STATE_VALVE_CLOSING;
END_IF;

STATE_VALVE_CLOSING: (* Закрытие клапана. *)
Timer1     := Timer1 + Ts_ms;
StateOpen  := FALSE;
StateClose := FALSE;
Error      := FALSE;
(* Если доехали до датчика то переходим в состояние закрыто. *)
(* Если нет обратной связи по датчику то переходим в состояние закрыто по таймеру. *)
IF (FeedbackClose OR (NOT(OnFeedbackClose) AND (Timer1>=TimeClose)) ) THEN
State1 := STATE_VALVE_CLOSE;
END_IF;
(* Если клапан заклинил и не доехал до датчика за заданное время уходим в состояние ошибки. *)
IF (OnFeedbackClose AND (Timer1>=TimeClose) ) THEN
State1 := STATE_ERROR_CLOSE;
END_IF;
(* Если во время закрытия пришла команда на открытие переходим в режим открытие. *)
IF (CommandOpen) THEN
State1 := STATE_VALVE_OPENING;
END_IF;

STATE_VALVE_CLOSE: (* Клапан закрыт. *)
Timer1     := 0;
StateOpen  := FALSE;
StateClose := TRUE;
Error      := FALSE;
(* Если пришла команда на открытие то переходим в состояние открытие. *)
IF (CommandOpen) THEN
State1 := STATE_VALVE_OPENING;
END_IF;

STATE_VALVE_OPENING: (* Открытие клапана. *)
Timer1     := Timer1 + Ts_ms;
StateOpen  := FALSE;
StateClose := FALSE;
Error      := FALSE;
(* Если доехали до датчика то переходим в состояние открыто. *)
(* Если нет обратной связи по датчику то переходим в состояние открыто по таймеру. *)
IF (FeedbackOpen OR (NOT(OnFeedbackOpen) AND (Timer1>=TimeOpen)) ) THEN
State1 := STATE_VALVE_OPEN;
END_IF;
(* Если клапан заклинил и не доехал до датчика за заданное время уходим в состояние ошибки. *)
IF (OnFeedbackOpen AND (Timer1>=TimeOpen) ) THEN
State1 := STATE_ERROR_OPEN;
END_IF;
(* Если во время открытия пришла команда на закрытие переходим в режим закрытие. *)
IF NOT(CommandOpen) THEN
State1 := STATE_VALVE_CLOSING;
END_IF;

STATE_VALVE_OPEN: (* Клапан открыт. *)
Timer1     := 0;
StateOpen  := TRUE;
StateClose := FALSE;
Error      := FALSE;
(* Если пришла команда на закрытие то переходим в состояние закрытие. *)
IF NOT(CommandOpen) THEN
State1 := STATE_VALVE_CLOSING;
END_IF;

STATE_ERROR_CLOSE: (* Клапан не закрылся. *)
Timer1     := 0;
StateOpen  := FALSE;
StateClose := FALSE;
Error      := TRUE;
(* Если все таки доехали до датчика то сброс для перехода на правильное состояние. *)
(* Если пришла команда на отрытие то сброс для перехода на правильное состояние. *)
(* Если выключили контроль обратной связи то сброс для перехода на правильное состояние. *)
IF (FeedbackClose OR CommandOpen OR NOT(OnFeedbackClose)) THEN
State1 := STATE_RESET;
END_IF;

STATE_ERROR_OPEN: (* Клапан не открылся. *)
Timer1     := 0;
StateOpen  := FALSE;
StateClose := FALSE;
Error      := TRUE;
(* Если все таки доехали до датчика то сброс для перехода на правильное состояние. *)
(* Если пришла команда на закрытие то сброс для перехода на правильное состояние. *)
(* Если выключили контроль обратной связи то сброс для перехода на правильное состояние. *)
IF (FeedbackOpen OR NOT(CommandOpen) OR NOT(OnFeedbackOpen)) THEN
State1 := STATE_RESET;
END_IF;

ELSE (* СТОП при неопределенном состоянии. *)
State1 := STATE_RESET;
END_CASE;

(*
@COPYLEFT ALL WRONGS RESERVED :)
Author: VA
Contacts: DIY.PLC.314@gmail.com
Date start LIB_PLC: 2014
License: GNU GPL-2.0-or-later
https://www.gnu.org/licenses/old-licenses/gpl-2.0.html
https://www.youtube.com/watch?v=n1F_MfLRlX0
https://www.youtube.com/@DIY_PLC
https://github.com/DIYPLC/LIB_PLC
https://oshwlab.com/diy.plc.314/PLC_HW1_SW1
https://3dtoday.ru/3d-models/mechanical-parts/body/korpus-na-din-reiku
https://t.me/DIY_PLC
*)
END_FUNCTION_BLOCK
